// TIA Portal V19 export
TYPE "C106_VAR_IF_NET_TYPIC"
   STRUCT
      BSC1 { ExternalAccessible := 'False'; ExternalVisible := 'False'; ExternalWritable := 'False'} : Bool;   // Netaansluiting beschikbaar
      BSC2 { ExternalAccessible := 'False'; ExternalVisible := 'False'; ExternalWritable := 'False'} : Bool;   // Netaansluiting niet beschikbaar
      BSC3 { ExternalAccessible := 'False'; ExternalVisible := 'False'; ExternalWritable := 'False'} : Bool;   // Netaansluiting beperkt beschikbaar
      STS_KR { ExternalAccessible := 'False'; ExternalVisible := 'False'; ExternalWritable := 'False'} : Bool;   // Kritiek
      STS_GKR { ExternalAccessible := 'False'; ExternalVisible := 'False'; ExternalWritable := 'False'} : Bool;   // Gestopt kritiek
      TYD_GKR { ExternalAccessible := 'False'; ExternalVisible := 'False'; ExternalWritable := 'False'} : Real;   // Tijdverloop voor Gestopt Kritiek
      EXT_AUT { ExternalAccessible := 'False'; ExternalVisible := 'False'; ExternalWritable := 'False'} : Bool;   // Externe (hoofd) beveiliging aangesproken
      EXT_HW { ExternalAccessible := 'False'; ExternalVisible := 'False'; ExternalWritable := 'False'} : Bool;   // Sturings hardware (PLC) in storing
      STO { ExternalAccessible := 'False'; ExternalVisible := 'False'; ExternalWritable := 'False'} : Struct   // Opsomming van alle storingen
         A001 : Bool;   // Beveiliging aangesproken
         A002 : Bool;   // Netaansluiting in storing
         A003 : Bool;   // Algemene storing netaansluiting
         A004 : Bool;   // Geen netaansluiting beschikbaar
         A005 : Bool;   // NSA niet gestart na uitval netaansluiting
      END_STRUCT;
   END_STRUCT;
END_TYPE
